// TIA Portal V18 export
FUNCTION "FC_AnalogOutCoverter" : Void   // FC8, STL
{ S7_Optimized_Access := 'TRUE' }
VERSION : 0.1
// stored: AutoNumber true, UDAEnableTagReadback false
   VAR_INPUT
      in_AnalogData : Real;
      in_NormMax : Real;
      in_NormMin : Real;
   END_VAR
   VAR_OUTPUT
      out_AnalogData : Int;
   END_VAR
   VAR_TEMP
      normData : Real;
      retData : Word;
   END_VAR
BEGIN

NETWORK
TITLE = 
//Conversor de salidas analogicas
      CALL  NORM_X
      ( MIN     := #in_NormMin,
        VALUE   := #in_AnalogData,
        MAX     := #in_NormMax,
        Ret_Val := #normData
      );

      CALL  SCALE_X
      ( MIN     := 0,
        VALUE   := #normData,
        MAX     := 27648,
        Ret_Val := #out_AnalogData
      );


//Unipolar:0 a 27648 Bipolar:-27648 a 27648


END_FUNCTION
